FUNCTION_BLOCK SBCActorRC (* Combines the SBActor and SBCalibrator function blocks *)
  (* Standard: 61499-2; Description: Requires the http communication layer. This function block makes use of CLNTRC FBs (see Utils subdirectory of this library) instead of CLIENT FBs. *)
  (* Version 1.0, 2017-08-27, Marc Jakobi, HTW Berlin *)
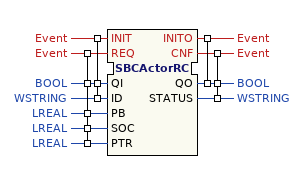
  EVENT_INPUT
    INIT WITH QI, ID; (* Initialization Request *)
    REQ WITH QI, PB, SOC, PTR; (* Normal Execution Request *)
  END_EVENT
  EVENT_OUTPUT
    INITO WITH QO; (* Initialization Confirm *)
    CNF WITH QO, STATUS; (* Execution Confirmation *)
  END_EVENT
  VAR_INPUT
    QI : BOOL; (* Input event qualifier *)
    ID : WSTRING; (* Connection identifier (ip:port) *)
    PB : LREAL; (* Battery transfer (positive = charge, negative = discharge) in W *)
    SOC : LREAL; (* State of charge [0,..,1] *)
    PTR : LREAL; (* Power used to release from trickle charge in W *)
  END_VAR
  VAR_OUTPUT
    QO : BOOL; (* Output event qualifier *)
    STATUS : WSTRING; (* HTTP response codes *)
  END_VAR
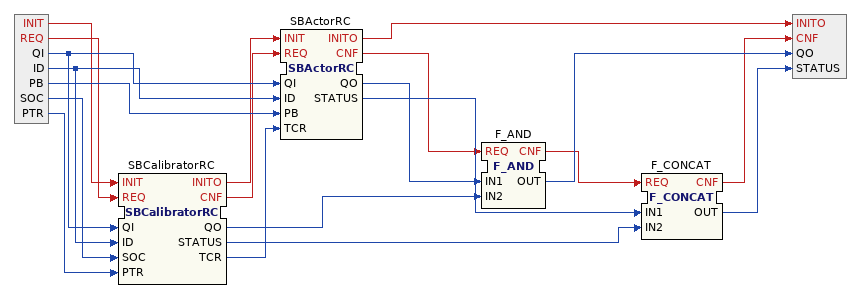
  FBS
    F_AND : F_AND;
    F_CONCAT : F_CONCAT;
    SBActorRC : SBActorRC;
    SBCalibratorRC : SBCalibratorRC;
  END_FBS
  EVENT_CONNECTIONS
    F_AND.CNF TO F_CONCAT.REQ;
    F_CONCAT.CNF TO CNF;
    SBActorRC.INITO TO INITO;
    SBActorRC.CNF TO F_AND.REQ;
    INIT TO SBCalibratorRC.INIT;
    REQ TO SBCalibratorRC.REQ;
    SBCalibratorRC.INITO TO SBActorRC.INIT;
    SBCalibratorRC.CNF TO SBActorRC.REQ;
  END_CONNECTIONS
  DATA_CONNECTIONS
    F_AND.OUT TO QO;
    F_CONCAT.OUT TO STATUS;
    QI TO SBActorRC.QI;
    ID TO SBActorRC.ID;
    PB TO SBActorRC.PB;
    SBActorRC.QO TO F_AND.IN1;
    SBActorRC.STATUS TO F_CONCAT.IN1;
    QI TO SBCalibratorRC.QI;
    ID TO SBCalibratorRC.ID;
    SOC TO SBCalibratorRC.SOC;
    PTR TO SBCalibratorRC.PTR;
    SBCalibratorRC.QO TO F_AND.IN2;
    SBCalibratorRC.STATUS TO F_CONCAT.IN2;
    SBCalibratorRC.TCR TO SBActorRC.TCR;
  END_CONNECTIONS
END_FUNCTION_BLOCK
